// TIA Portal V17 export
// export: Created 2024-09-02T12:50:05.3382635Z, ExportSetting WithDefaults, DisplayName Totally Integrated Automation Portal, DisplayVersion V17, DisplayName TIA Portal Openness, DisplayVersion V17, DisplayName TIA Portal Version Control Interface, DisplayVersion V17, DisplayName STEP 7 Professional, DisplayVersion V17, DisplayName STEP 7 Safety, DisplayVersion V17, DisplayName WinCC Professional, DisplayVersion V17
DATA_BLOCK "CPU Monitoring_DB"   // DB7
VERSION : 0.1
// stored: AutoNumber true, DBAccessibleFromOPCUA true, InstanceOfName CPU Monitoring, InstanceOfType FB
"CPU Monitoring"
   // VAR
   //    Mode : UInt;
   //    OBnr : OB_ANY;
   //    InfoData : UInt;
   //    ReturnValue : Int;
   // END_VAR
BEGIN
END_DATA_BLOCK
